PROGRAM MAIN
VAR
	nSwitchCtrl : BOOL := TRUE;
	nRotateUpper : WORD :=16#8000;
	nRotateLower :WORD :=16#01;
	bEL6224_Ch1 AT%I* : ARRAY[0..1] OF BYTE;
END_VAR

//SICK_Process_Parse(Data:=bEL6224_Ch1 , Process_Data=>GVL.SICK_1_Process );
GVL.SICK_1_Process := SICK_Process_Parse(Data:=bEL6224_Ch1);



























































































































]

END_PROGRAM

(* stored: Version 1.1.0.1, ProductVersion 3.1.4024.10
   POU MAIN: Id {fbf67ee1-36f3-4031-825a-38fcbb72130e}, SpecialFunc None *)
